// Mitsubishi GX Works2 project: GBOD-1507C(20080005)_210617up   PLC: Q03UDV

PROGRAM MAIN
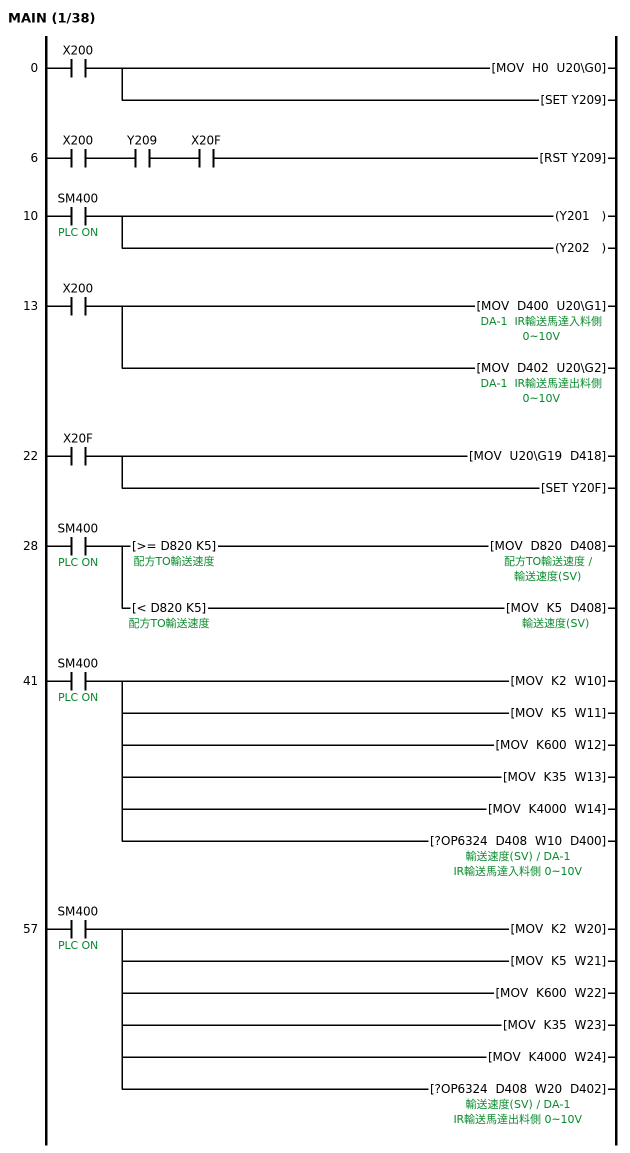
0     LD      X200
      MOV     H0 U20\G0
      SET     Y209
6     LD      X200
      AND     Y209
      AND     X20F
      RST     Y209
10    LD      SM400  ; PLC ON
      OUT     Y201
      OUT     Y202
13    LD      X200
      MOV     D400 U20\G1  ; DA-1  IR輸送馬達入料側 0~10V
      MOV     D402 U20\G2  ; DA-1  IR輸送馬達出料側 0~10V
22    LD      X20F
      MOV     U20\G19 D418
      SET     Y20F
28    LD      SM400  ; PLC ON
      MPS
      AND>=   D820 K5  ; 配方TO輸送速度
      MOV     D820 D408  ; 輸送速度(SV)
      MPP
      AND<    D820 K5  ; 配方TO輸送速度
      MOV     K5 D408
41    LD      SM400  ; PLC ON
      MOV     K2 W10
        [note] 
      MOV     K5 W11
      MOV     K600 W12
      MOV     K35 W13
      MOV     K4000 W14
      ?OP6324 D408 W10 D400
57    LD      SM400  ; PLC ON
      MOV     K2 W20
        [note] 
      MOV     K5 W21
      MOV     K600 W22
      MOV     K35 W23
      MOV     K4000 W24
      ?OP6324 D408 W20 D402
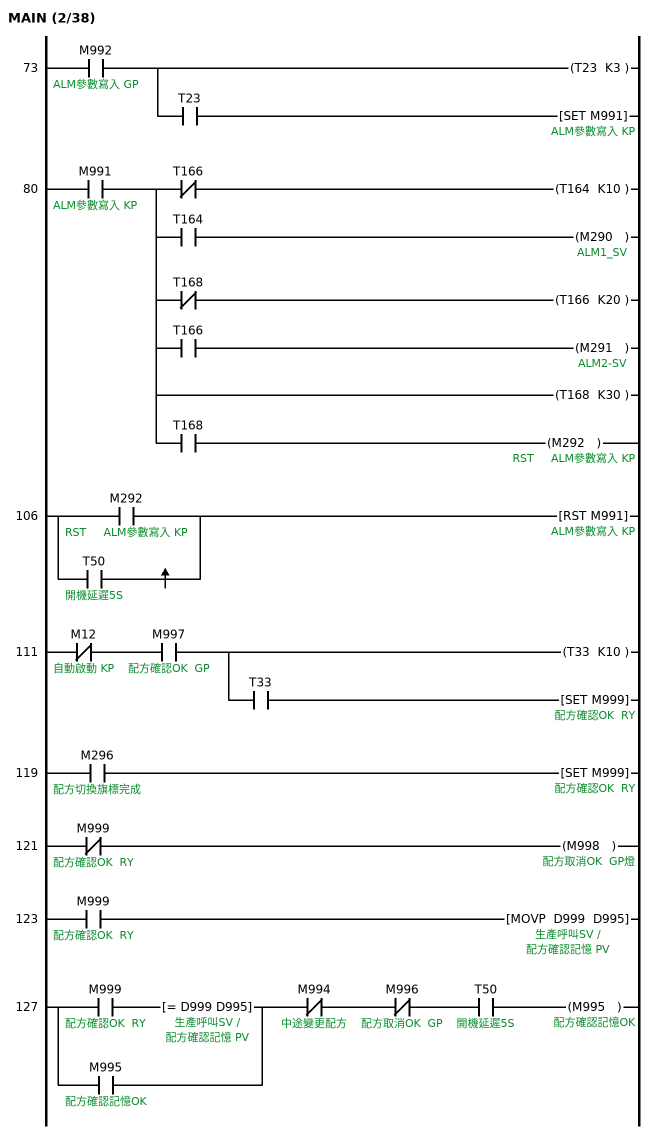
73    LD      M992  ; ALM參數寫入 GP
      OUT     T23 K3
      AND     T23
      SET     M991  ; ALM參數寫入 KP
80    LD      M991  ; ALM參數寫入 KP
      MPS
      ANI     T166
      OUT     T164 K10
      MRD
      AND     T164
      OUT     M290  ; ALM1_SV
      MRD
      ANI     T168
      OUT     T166 K20
      MRD
      AND     T166
      OUT     M291  ; ALM2-SV
      MPP
      OUT     T168 K30
      AND     T168
      OUT     M292  ; RST     ALM參數寫入 KP
106   LD      M292  ; RST     ALM參數寫入 KP
      LD      T50  ; 開機延遲5S
      MEP
      ORB
      RST     M991  ; ALM參數寫入 KP
111   LDI     M12  ; 自動啟動 KP
      AND     M997  ; 配方確認OK  GP
      OUT     T33 K10
      AND     T33
      SET     M999  ; 配方確認OK  RY
119   LD      M296  ; 配方切換旗標完成
      SET     M999  ; 配方確認OK  RY
121   LDI     M999  ; 配方確認OK  RY
      OUT     M998  ; 配方取消OK  GP燈
123   LD      M999  ; 配方確認OK  RY
      MOVP    D999 D995  ; 生產呼叫SV / 配方確認記憶 PV
127   LD      M999  ; 配方確認OK  RY
      AND=    D999 D995  ; 生產呼叫SV / 配方確認記憶 PV
      OR      M995  ; 配方確認記憶OK
      ANI     M994  ; 中途變更配方
      ANI     M996  ; 配方取消OK  GP
      AND     T50  ; 開機延遲5S
      OUT     M995  ; 配方確認記憶OK
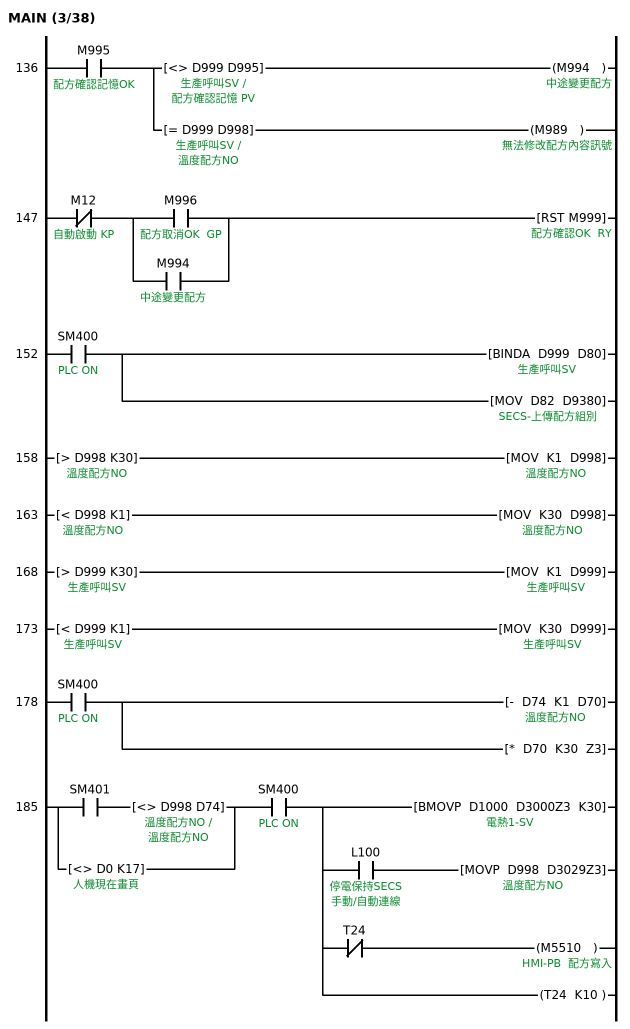
136   LD      M995  ; 配方確認記憶OK
      MPS
      AND<>   D999 D995  ; 生產呼叫SV / 配方確認記憶 PV
      OUT     M994  ; 中途變更配方
      MPP
      AND=    D999 D998  ; 生產呼叫SV / 溫度配方NO
      OUT     M989  ; 無法修改配方內容訊號
147   LDI     M12  ; 自動啟動 KP
      LD      M996  ; 配方取消OK  GP
      OR      M994  ; 中途變更配方
      ANB
      RST     M999  ; 配方確認OK  RY
152   LD      SM400  ; PLC ON
      BINDA   D999 D80
      MOV     D82 D9380  ; SECS-上傳配方組別
158   LD>     D998 K30  ; 溫度配方NO
      MOV     K1 D998
163   LD<     D998 K1  ; 溫度配方NO
      MOV     K30 D998
168   LD>     D999 K30  ; 生產呼叫SV
      MOV     K1 D999
173   LD<     D999 K1  ; 生產呼叫SV
      MOV     K30 D999
178   LD      SM400  ; PLC ON
      -       D74 K1 D70  ; 溫度配方NO
      *       D70 K30 Z3
185   LD      SM401
      AND<>   D998 D74  ; 溫度配方NO / 溫度配方NO
      OR<>    D0 K17  ; 人機現在畫頁
      AND     SM400  ; PLC ON
      BMOVP   D1000 D3000Z3 K30  ; 電熱1-SV
      MPS
      AND     L100  ; 停電保持SECS    手動/自動連線
      MOVP    D998 D3029Z3
      MRD
      ANI     T24
      OUT     M5510  ; HMI-PB  配方寫入
      MPP
      OUT     T24 K10
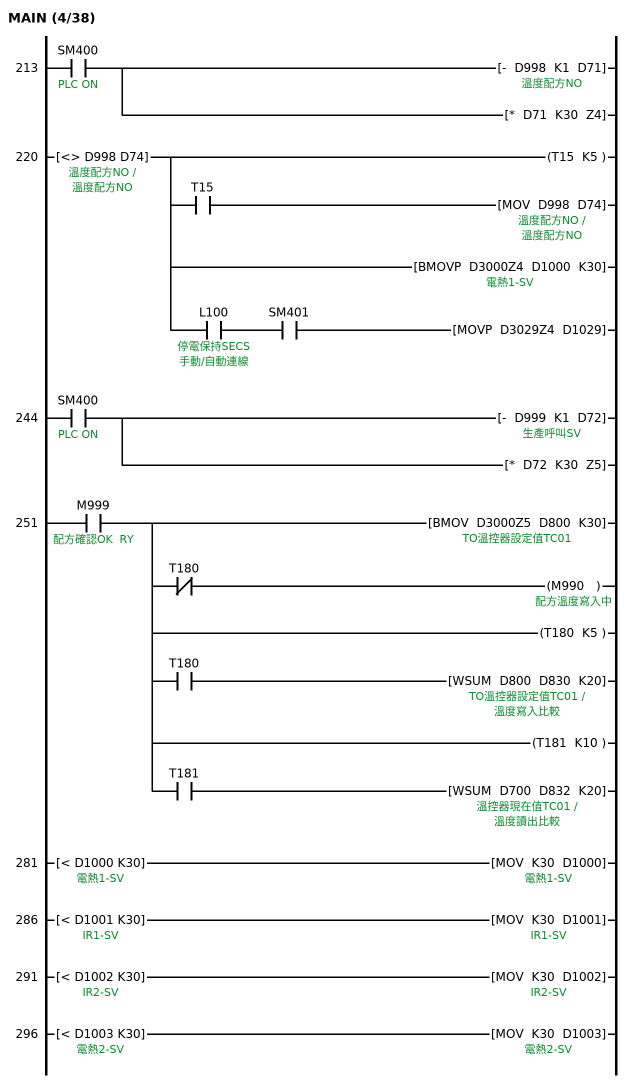
213   LD      SM400  ; PLC ON
      -       D998 K1 D71
      *       D71 K30 Z4
220   LD<>    D998 D74  ; 溫度配方NO / 溫度配方NO
      OUT     T15 K5
      MPS
      AND     T15
      MOV     D998 D74
      MPP
      BMOVP   D3000Z4 D1000 K30
      AND     L100  ; 停電保持SECS    手動/自動連線
      AND     SM401
      MOVP    D3029Z4 D1029
244   LD      SM400  ; PLC ON
      -       D999 K1 D72
      *       D72 K30 Z5
251   LD      M999  ; 配方確認OK  RY
      BMOV    D3000Z5 D800 K30  ; TO溫控器設定值TC01
      MPS
      ANI     T180
      OUT     M990  ; 配方溫度寫入中
      MPP
      OUT     T180 K5
      MPS
      AND     T180
      WSUM    D800 D830 K20  ; 溫度寫入比較
      MPP
      OUT     T181 K10
      AND     T181
      WSUM    D700 D832 K20  ; 溫控器現在值TC01 / 溫度讀出比較
281   LD<     D1000 K30  ; 電熱1-SV
      MOV     K30 D1000
286   LD<     D1001 K30  ; IR1-SV
      MOV     K30 D1001
291   LD<     D1002 K30  ; IR2-SV
      MOV     K30 D1002
296   LD<     D1003 K30  ; 電熱2-SV
      MOV     K30 D1003
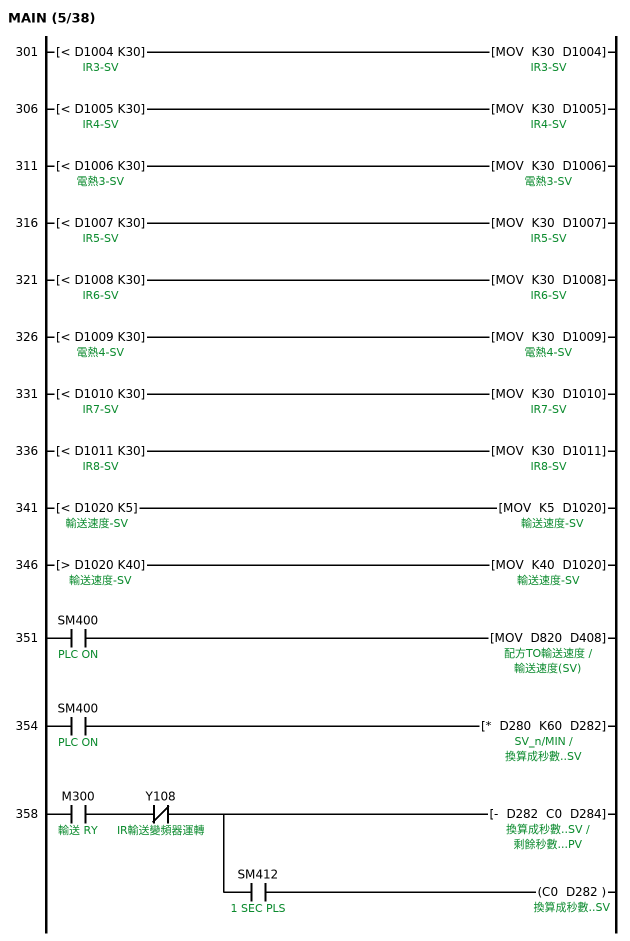
301   LD<     D1004 K30  ; IR3-SV
      MOV     K30 D1004
306   LD<     D1005 K30  ; IR4-SV
      MOV     K30 D1005
311   LD<     D1006 K30  ; 電熱3-SV
      MOV     K30 D1006
316   LD<     D1007 K30  ; IR5-SV
      MOV     K30 D1007
321   LD<     D1008 K30  ; IR6-SV
      MOV     K30 D1008
326   LD<     D1009 K30  ; 電熱4-SV
      MOV     K30 D1009
331   LD<     D1010 K30  ; IR7-SV
      MOV     K30 D1010
336   LD<     D1011 K30  ; IR8-SV
      MOV     K30 D1011
341   LD<     D1020 K5  ; 輸送速度-SV
      MOV     K5 D1020
346   LD>     D1020 K40  ; 輸送速度-SV
      MOV     K40 D1020
351   LD      SM400  ; PLC ON
      MOV     D820 D408
354   LD      SM400  ; PLC ON
      *       D280 K60 D282  ; SV_n/MIN / 換算成秒數..SV
358   LD      M300  ; 輸送 RY
      ANI     Y108  ; IR輸送變頻器運轉
      -       D282 C0 D284  ; 剩餘秒數...PV
      AND     SM412  ; 1 SEC PLS
      OUT     C0 D282  ; 換算成秒數..SV
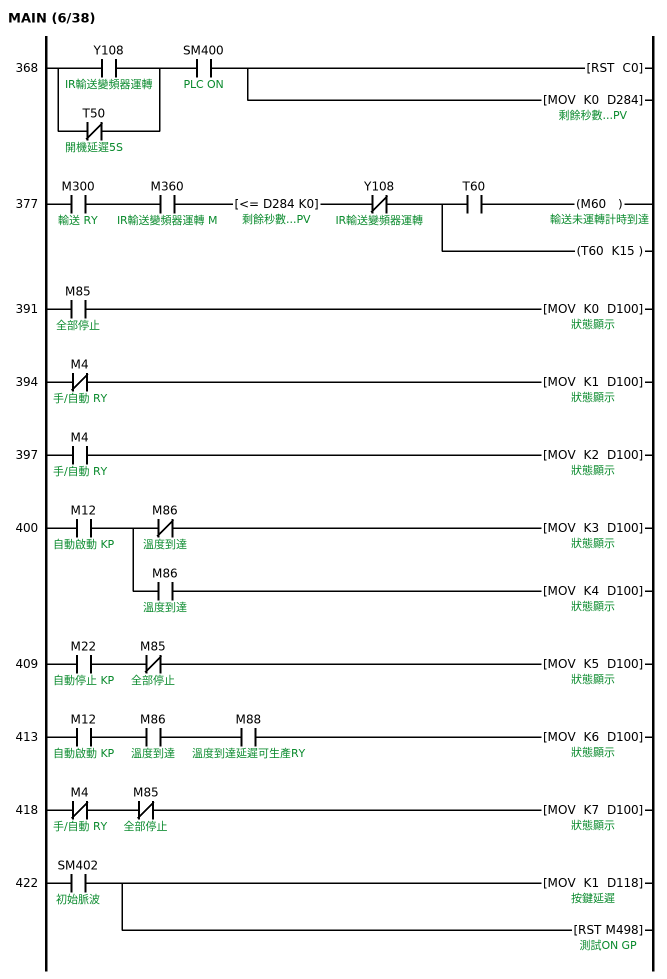
368   LD      Y108  ; IR輸送變頻器運轉
      ORI     T50  ; 開機延遲5S
      AND     SM400  ; PLC ON
      RST     C0
      MOV     K0 D284
377   LD      M300  ; 輸送 RY
      AND     M360  ; IR輸送變頻器運轉 M
      AND<=   D284 K0  ; 剩餘秒數...PV
      ANI     Y108  ; IR輸送變頻器運轉
      MPS
      AND     T60
      OUT     M60  ; 輸送未運轉計時到達
      MPP
      OUT     T60 K15
391   LD      M85  ; 全部停止
      MOV     K0 D100  ; 狀態顯示
394   LDI     M4  ; 手/自動 RY
      MOV     K1 D100
397   LD      M4  ; 手/自動 RY
      MOV     K2 D100
400   LD      M12  ; 自動啟動 KP
      MPS
      ANI     M86  ; 溫度到達
      MOV     K3 D100
      MPP
      AND     M86  ; 溫度到達
      MOV     K4 D100
409   LD      M22  ; 自動停止 KP
      ANI     M85  ; 全部停止
      MOV     K5 D100
413   LD      M12  ; 自動啟動 KP
      AND     M86  ; 溫度到達
      AND     M88  ; 溫度到達延遲可生產RY
      MOV     K6 D100
418   LDI     M4  ; 手/自動 RY
      ANI     M85  ; 全部停止
      MOV     K7 D100
422   LD      SM402  ; 初始脈波
      MOV     K1 D118  ; 按鍵延遲
      RST     M498  ; 測試ON GP
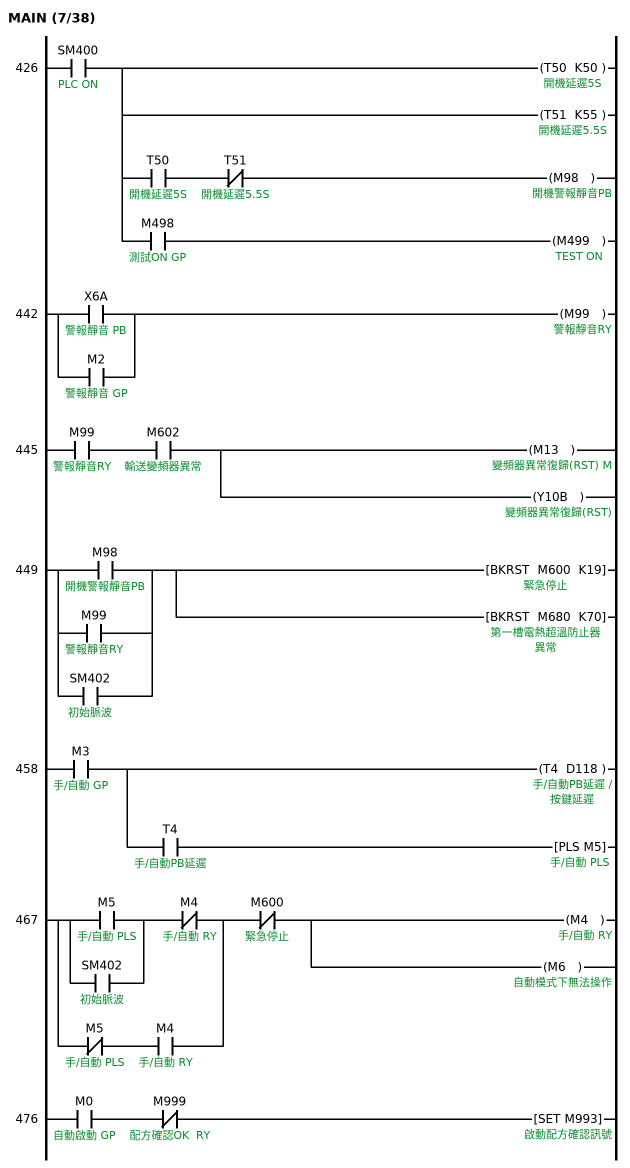
426   LD      SM400  ; PLC ON
      OUT     T50 K50  ; 開機延遲5S
      OUT     T51 K55  ; 開機延遲5.5S
      MPS
      AND     T50  ; 開機延遲5S
      ANI     T51  ; 開機延遲5.5S
      OUT     M98  ; 開機警報靜音PB
      MPP
      AND     M498  ; 測試ON GP
      OUT     M499  ; TEST ON
442   LD      X6A  ; 警報靜音 PB
      OR      M2  ; 警報靜音 GP
      OUT     M99  ; 警報靜音RY
445   LD      M99  ; 警報靜音RY
      AND     M602  ; 輸送變頻器異常
      OUT     M13  ; 變頻器異常復歸(RST) M
      OUT     Y10B  ; 變頻器異常復歸(RST)
449   LD      M98  ; 開機警報靜音PB
      OR      M99  ; 警報靜音RY
      OR      SM402  ; 初始脈波
      BKRST   M600 K19  ; 緊急停止
      BKRST   M680 K70  ; 第一槽電熱超溫防止器異常
458   LD      M3  ; 手/自動 GP
      OUT     T4 D118  ; 手/自動PB延遲 / 按鍵延遲
        [note] 
      AND     T4  ; 手/自動PB延遲
      PLS     M5  ; 手/自動 PLS
467   LD      M5  ; 手/自動 PLS
      OR      SM402  ; 初始脈波
      ANI     M4  ; 手/自動 RY
      LDI     M5  ; 手/自動 PLS
      AND     M4  ; 手/自動 RY
      ORB
      ANI     M600  ; 緊急停止
      OUT     M4  ; 手/自動 RY
      OUT     M6  ; 自動模式下無法操作
476   LD      M0  ; 自動啟動 GP
      ANI     M999  ; 配方確認OK  RY
      SET     M993  ; 啟動配方確認訊號
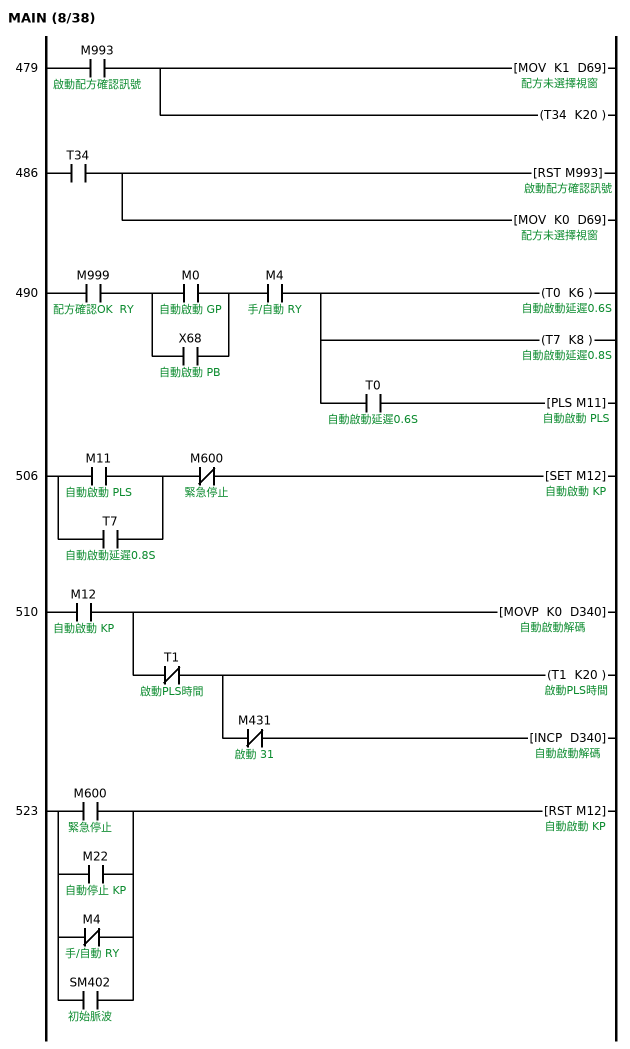
479   LD      M993  ; 啟動配方確認訊號
      MOV     K1 D69  ; 配方未選擇視窗
      OUT     T34 K20
486   LD      T34
      RST     M993  ; 啟動配方確認訊號
      MOV     K0 D69
490   LD      M999  ; 配方確認OK  RY
      LD      M0  ; 自動啟動 GP
      OR      X68  ; 自動啟動 PB
      ANB
      AND     M4  ; 手/自動 RY
      OUT     T0 K6  ; 自動啟動延遲0.6S
      OUT     T7 K8  ; 自動啟動延遲0.8S
      AND     T0  ; 自動啟動延遲0.6S
      PLS     M11  ; 自動啟動 PLS
506   LD      M11  ; 自動啟動 PLS
      OR      T7  ; 自動啟動延遲0.8S
      ANI     M600  ; 緊急停止
      SET     M12  ; 自動啟動 KP
510   LD      M12  ; 自動啟動 KP
      MOVP    K0 D340  ; 自動啟動解碼
      ANI     T1  ; 啟動PLS時間
      OUT     T1 K20  ; 啟動PLS時間
      ANI     M431  ; 啟動 31
      INCP    D340
523   LD      M600  ; 緊急停止
      OR      M22  ; 自動停止 KP
      ORI     M4  ; 手/自動 RY
      OR      SM402  ; 初始脈波
      RST     M12  ; 自動啟動 KP
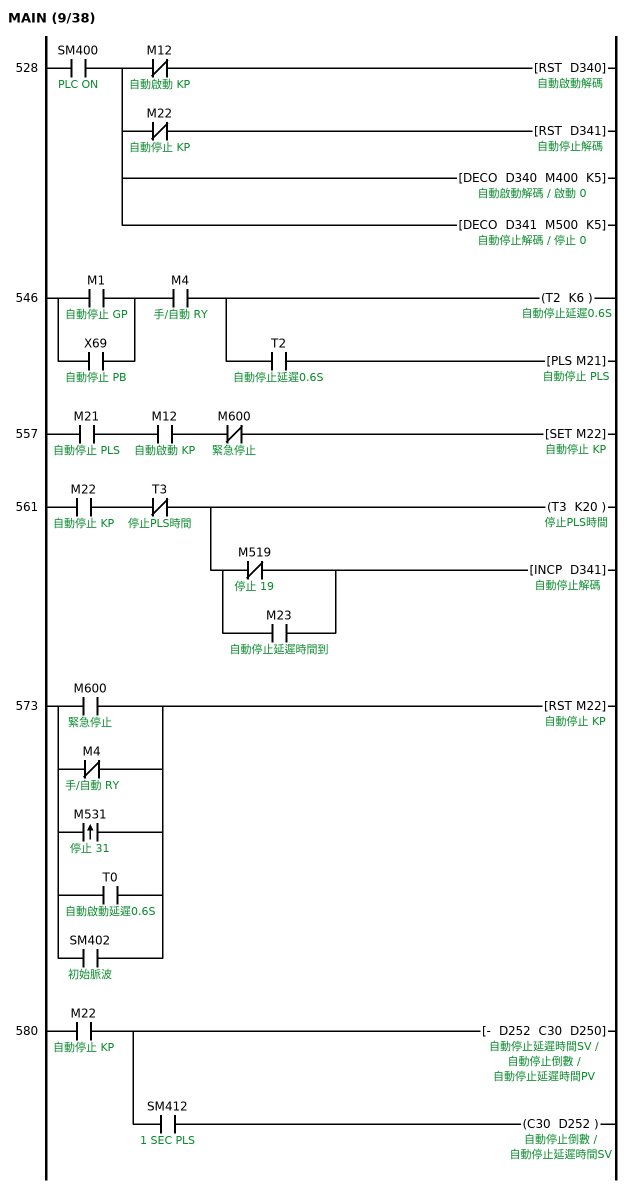
528   LD      SM400  ; PLC ON
      MPS
      ANI     M12  ; 自動啟動 KP
      RST     D340  ; 自動啟動解碼
      MRD
      ANI     M22  ; 自動停止 KP
      RST     D341  ; 自動停止解碼
      MPP
      DECO    D340 M400 K5  ; 啟動 0
      DECO    D341 M500 K5  ; 停止 0
546   LD      M1  ; 自動停止 GP
      OR      X69  ; 自動停止 PB
      AND     M4  ; 手/自動 RY
      OUT     T2 K6  ; 自動停止延遲0.6S
        [note] 
      AND     T2  ; 自動停止延遲0.6S
      PLS     M21  ; 自動停止 PLS
557   LD      M21  ; 自動停止 PLS
      AND     M12  ; 自動啟動 KP
      ANI     M600  ; 緊急停止
      SET     M22  ; 自動停止 KP
561   LD      M22  ; 自動停止 KP
      ANI     T3  ; 停止PLS時間
      OUT     T3 K20  ; 停止PLS時間
      LDI     M519  ; 停止 19
      OR      M23  ; 自動停止延遲時間到
      ANB
      INCP    D341
573   LD      M600  ; 緊急停止
      ORI     M4  ; 手/自動 RY
      ORP     M531  ; 停止 31
      OR      T0  ; 自動啟動延遲0.6S
      OR      SM402  ; 初始脈波
      RST     M22  ; 自動停止 KP
580   LD      M22  ; 自動停止 KP
      -       D252 C30 D250  ; 自動停止延遲時間SV / 自動停止倒數 / 自動停止延遲時間PV
      AND     SM412  ; 1 SEC PLS
      OUT     C30 D252  ; 自動停止倒數 / 自動停止延遲時間SV
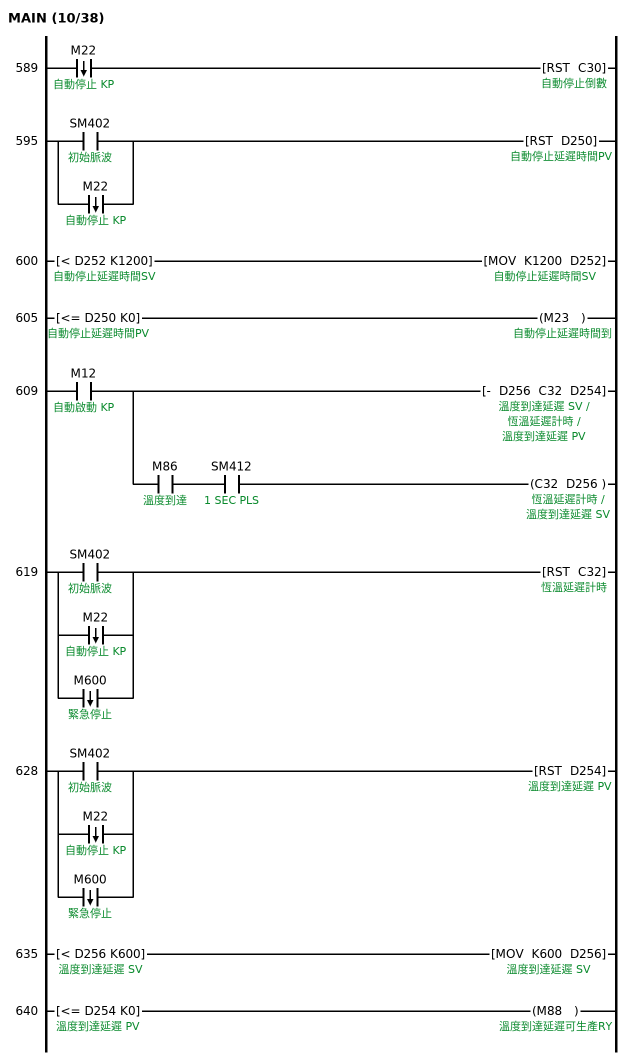
589   LDF     M22  ; 自動停止 KP
      RST     C30  ; 自動停止倒數
595   LD      SM402  ; 初始脈波
      ORF     M22  ; 自動停止 KP
      RST     D250  ; 自動停止延遲時間PV
600   LD<     D252 K1200  ; 自動停止延遲時間SV
      MOV     K1200 D252
605   LD<=    D250 K0  ; 自動停止延遲時間PV
      OUT     M23  ; 自動停止延遲時間到
609   LD      M12  ; 自動啟動 KP
      -       D256 C32 D254  ; 溫度到達延遲 SV / 恆溫延遲計時 / 溫度到達延遲 PV
      AND     M86  ; 溫度到達
      AND     SM412  ; 1 SEC PLS
      OUT     C32 D256  ; 恆溫延遲計時 / 溫度到達延遲 SV
619   LD      SM402  ; 初始脈波
      ORF     M22  ; 自動停止 KP
      ORF     M600  ; 緊急停止
      RST     C32  ; 恆溫延遲計時
628   LD      SM402  ; 初始脈波
      ORF     M22  ; 自動停止 KP
      ORF     M600  ; 緊急停止
      RST     D254  ; 溫度到達延遲 PV
635   LD<     D256 K600  ; 溫度到達延遲 SV
      MOV     K600 D256
640   LD<=    D254 K0  ; 溫度到達延遲 PV
      OUT     M88  ; 溫度到達延遲可生產RY
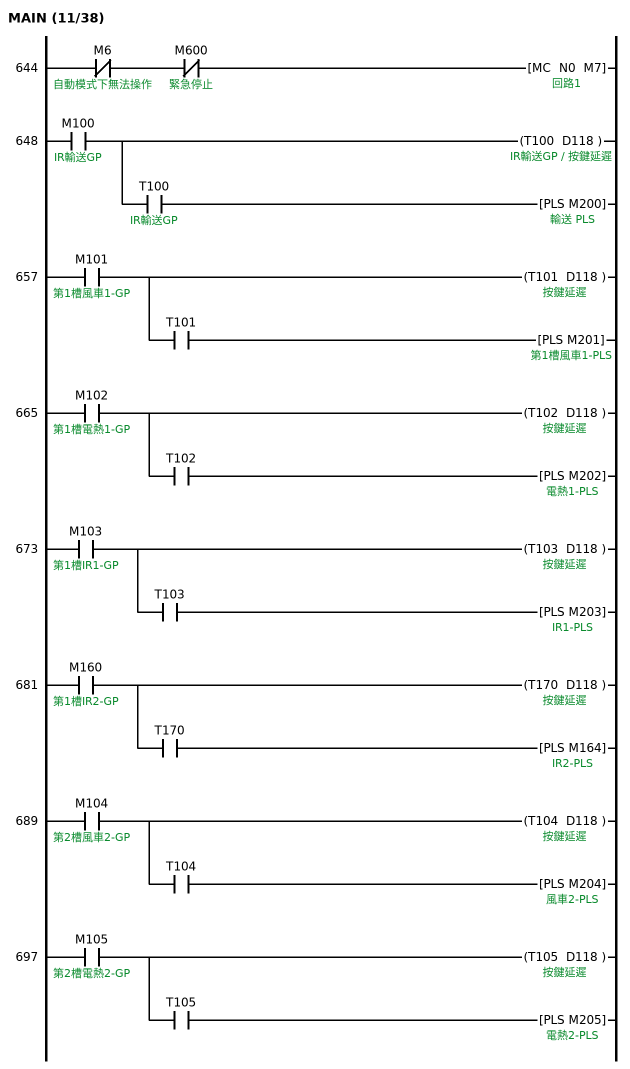
644   LDI     M6  ; 自動模式下無法操作
      ANI     M600  ; 緊急停止
      MC      N0 M7  ; 回路1
648   LD      M100  ; IR輸送GP
      OUT     T100 D118  ; IR輸送GP / 按鍵延遲
        [note] 
      AND     T100  ; IR輸送GP
      PLS     M200  ; 輸送 PLS
657   LD      M101  ; 第1槽風車1-GP
      OUT     T101 D118  ; 按鍵延遲
      AND     T101
      PLS     M201  ; 第1槽風車1-PLS
665   LD      M102  ; 第1槽電熱1-GP
      OUT     T102 D118  ; 按鍵延遲
      AND     T102
      PLS     M202  ; 電熱1-PLS
673   LD      M103  ; 第1槽IR1-GP
      OUT     T103 D118  ; 按鍵延遲
      AND     T103
      PLS     M203  ; IR1-PLS
681   LD      M160  ; 第1槽IR2-GP
      OUT     T170 D118  ; 按鍵延遲
      AND     T170
      PLS     M164  ; IR2-PLS
689   LD      M104  ; 第2槽風車2-GP
      OUT     T104 D118  ; 按鍵延遲
      AND     T104
      PLS     M204  ; 風車2-PLS
697   LD      M105  ; 第2槽電熱2-GP
      OUT     T105 D118  ; 按鍵延遲
      AND     T105
      PLS     M205  ; 電熱2-PLS
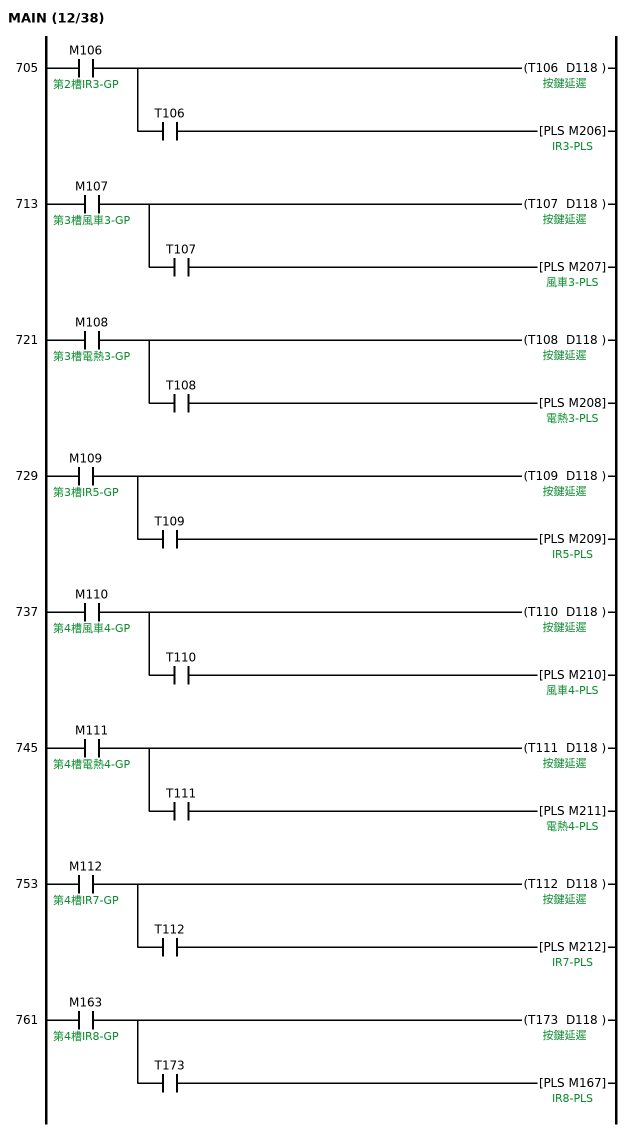
705   LD      M106  ; 第2槽IR3-GP
      OUT     T106 D118  ; 按鍵延遲
      AND     T106
      PLS     M206  ; IR3-PLS
713   LD      M107  ; 第3槽風車3-GP
      OUT     T107 D118  ; 按鍵延遲
      AND     T107
      PLS     M207  ; 風車3-PLS
721   LD      M108  ; 第3槽電熱3-GP
      OUT     T108 D118  ; 按鍵延遲
      AND     T108
      PLS     M208  ; 電熱3-PLS
729   LD      M109  ; 第3槽IR5-GP
      OUT     T109 D118  ; 按鍵延遲
      AND     T109
      PLS     M209  ; IR5-PLS
737   LD      M110  ; 第4槽風車4-GP
      OUT     T110 D118  ; 按鍵延遲
      AND     T110
      PLS     M210  ; 風車4-PLS
745   LD      M111  ; 第4槽電熱4-GP
      OUT     T111 D118  ; 按鍵延遲
      AND     T111
      PLS     M211  ; 電熱4-PLS
753   LD      M112  ; 第4槽IR7-GP
      OUT     T112 D118  ; 按鍵延遲
      AND     T112
      PLS     M212  ; IR7-PLS
761   LD      M163  ; 第4槽IR8-GP
      OUT     T173 D118  ; 按鍵延遲
      AND     T173
      PLS     M167  ; IR8-PLS
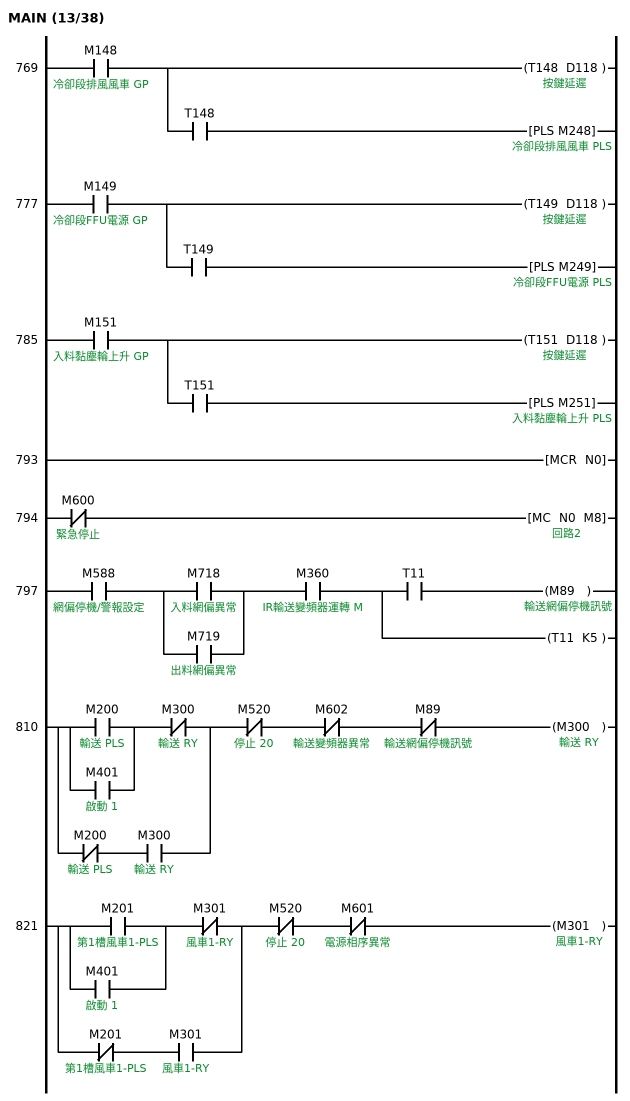
769   LD      M148  ; 冷卻段排風風車 GP
      OUT     T148 D118  ; 按鍵延遲
      AND     T148
      PLS     M248  ; 冷卻段排風風車 PLS
777   LD      M149  ; 冷卻段FFU電源 GP
      OUT     T149 D118  ; 按鍵延遲
      AND     T149
      PLS     M249  ; 冷卻段FFU電源 PLS
785   LD      M151  ; 入料黏塵輪上升 GP
      OUT     T151 D118  ; 按鍵延遲
      AND     T151
      PLS     M251  ; 入料黏塵輪上升 PLS
793   MCR     N0
794   LDI     M600  ; 緊急停止
      MC      N0 M8  ; 回路2
797   LD      M588  ; 網偏停機/警報設定
      LD      M718  ; 入料網偏異常
      OR      M719  ; 出料網偏異常
      ANB
      AND     M360  ; IR輸送變頻器運轉 M
      MPS
      AND     T11
      OUT     M89  ; 輸送網偏停機訊號
      MPP
      OUT     T11 K5
810   LD      M200  ; 輸送 PLS
      OR      M401  ; 啟動 1
      ANI     M300  ; 輸送 RY
      LDI     M200  ; 輸送 PLS
      AND     M300  ; 輸送 RY
      ORB
      ANI     M520  ; 停止 20
      ANI     M602  ; 輸送變頻器異常
      ANI     M89  ; 輸送網偏停機訊號
      OUT     M300  ; 輸送 RY
        [note] 
821   LD      M201  ; 第1槽風車1-PLS
      OR      M401  ; 啟動 1
      ANI     M301  ; 風車1-RY
      LDI     M201  ; 第1槽風車1-PLS
      AND     M301  ; 風車1-RY
      ORB
      ANI     M520  ; 停止 20
      ANI     M601  ; 電源相序異常
      OUT     M301  ; 風車1-RY
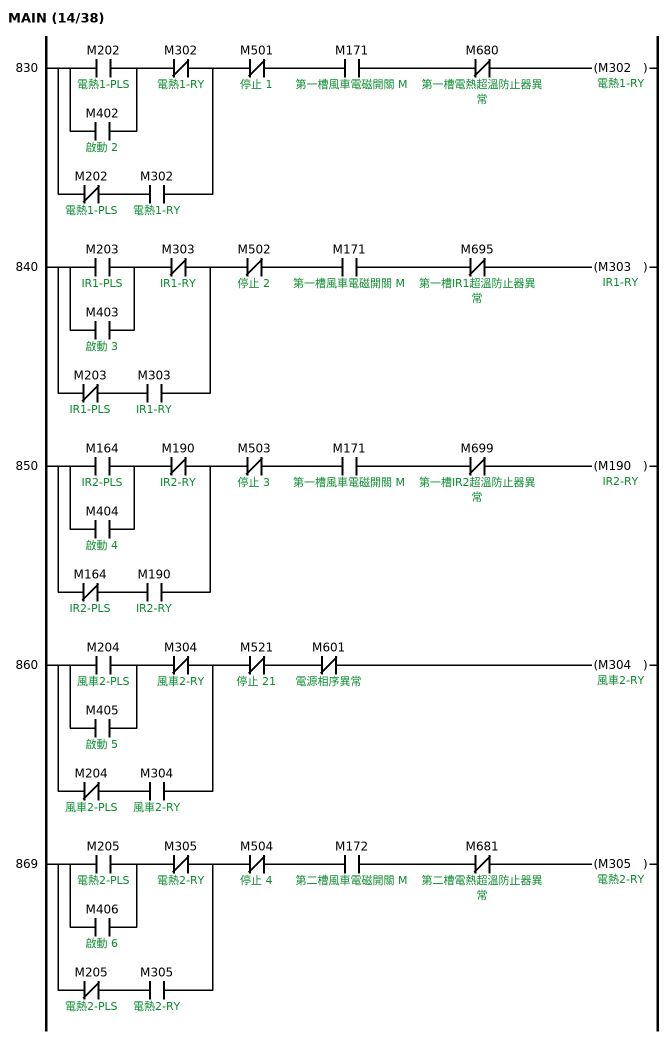
830   LD      M202  ; 電熱1-PLS
      OR      M402  ; 啟動 2
      ANI     M302  ; 電熱1-RY
      LDI     M202  ; 電熱1-PLS
      AND     M302  ; 電熱1-RY
      ORB
      ANI     M501  ; 停止 1
      AND     M171  ; 第一槽風車電磁開關 M
      ANI     M680  ; 第一槽電熱超溫防止器異常
      OUT     M302  ; 電熱1-RY
840   LD      M203  ; IR1-PLS
      OR      M403  ; 啟動 3
      ANI     M303  ; IR1-RY
      LDI     M203  ; IR1-PLS
      AND     M303  ; IR1-RY
      ORB
      ANI     M502  ; 停止 2
      AND     M171  ; 第一槽風車電磁開關 M
      ANI     M695  ; 第一槽IR1超溫防止器異常
      OUT     M303  ; IR1-RY
850   LD      M164  ; IR2-PLS
      OR      M404  ; 啟動 4
      ANI     M190  ; IR2-RY
      LDI     M164  ; IR2-PLS
      AND     M190  ; IR2-RY
      ORB
      ANI     M503  ; 停止 3
      AND     M171  ; 第一槽風車電磁開關 M
      ANI     M699  ; 第一槽IR2超溫防止器異常
      OUT     M190  ; IR2-RY
860   LD      M204  ; 風車2-PLS
      OR      M405  ; 啟動 5
      ANI     M304  ; 風車2-RY
      LDI     M204  ; 風車2-PLS
      AND     M304  ; 風車2-RY
      ORB
      ANI     M521  ; 停止 21
      ANI     M601  ; 電源相序異常
      OUT     M304  ; 風車2-RY
869   LD      M205  ; 電熱2-PLS
      OR      M406  ; 啟動 6
      ANI     M305  ; 電熱2-RY
      LDI     M205  ; 電熱2-PLS
      AND     M305  ; 電熱2-RY
      ORB
      ANI     M504  ; 停止 4
      AND     M172  ; 第二槽風車電磁開關 M
      ANI     M681  ; 第二槽電熱超溫防止器異常
      OUT     M305  ; 電熱2-RY
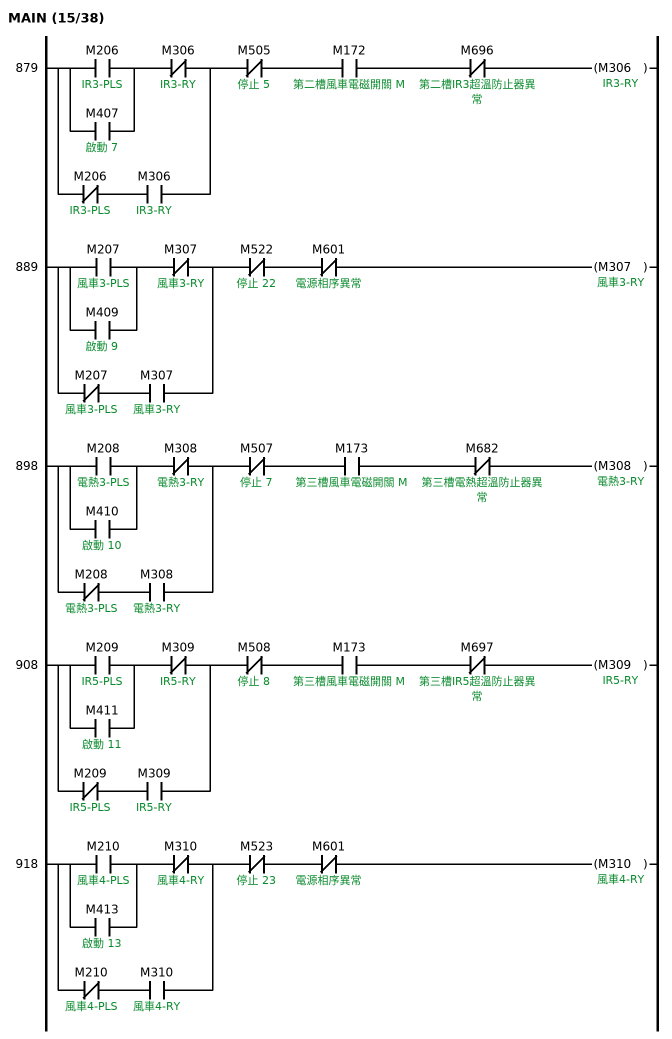
879   LD      M206  ; IR3-PLS
      OR      M407  ; 啟動 7
      ANI     M306  ; IR3-RY
      LDI     M206  ; IR3-PLS
      AND     M306  ; IR3-RY
      ORB
      ANI     M505  ; 停止 5
      AND     M172  ; 第二槽風車電磁開關 M
      ANI     M696  ; 第二槽IR3超溫防止器異常
      OUT     M306  ; IR3-RY
889   LD      M207  ; 風車3-PLS
      OR      M409  ; 啟動 9
      ANI     M307  ; 風車3-RY
      LDI     M207  ; 風車3-PLS
      AND     M307  ; 風車3-RY
      ORB
      ANI     M522  ; 停止 22
      ANI     M601  ; 電源相序異常
      OUT     M307  ; 風車3-RY
898   LD      M208  ; 電熱3-PLS
      OR      M410  ; 啟動 10
      ANI     M308  ; 電熱3-RY
      LDI     M208  ; 電熱3-PLS
      AND     M308  ; 電熱3-RY
      ORB
      ANI     M507  ; 停止 7
      AND     M173  ; 第三槽風車電磁開關 M
      ANI     M682  ; 第三槽電熱超溫防止器異常
      OUT     M308  ; 電熱3-RY
908   LD      M209  ; IR5-PLS
      OR      M411  ; 啟動 11
      ANI     M309  ; IR5-RY
      LDI     M209  ; IR5-PLS
      AND     M309  ; IR5-RY
      ORB
      ANI     M508  ; 停止 8
      AND     M173  ; 第三槽風車電磁開關 M
      ANI     M697  ; 第三槽IR5超溫防止器異常
      OUT     M309  ; IR5-RY
918   LD      M210  ; 風車4-PLS
      OR      M413  ; 啟動 13
      ANI     M310  ; 風車4-RY
      LDI     M210  ; 風車4-PLS
      AND     M310  ; 風車4-RY
      ORB
      ANI     M523  ; 停止 23
      ANI     M601  ; 電源相序異常
      OUT     M310  ; 風車4-RY
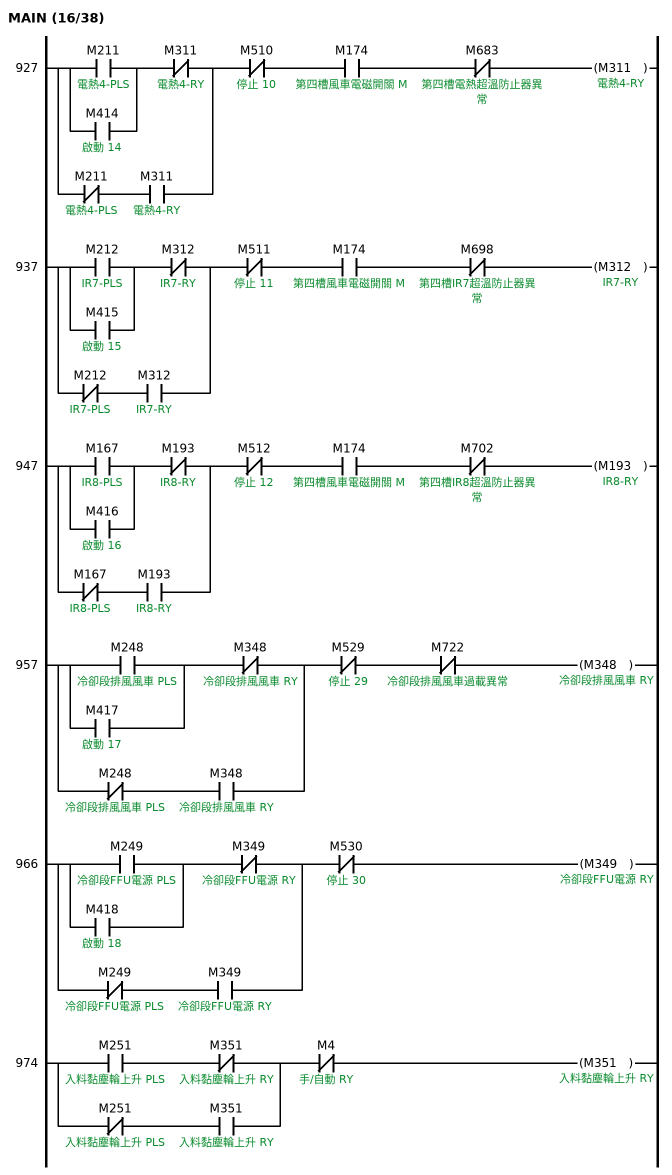
927   LD      M211  ; 電熱4-PLS
      OR      M414  ; 啟動 14
      ANI     M311  ; 電熱4-RY
      LDI     M211  ; 電熱4-PLS
      AND     M311  ; 電熱4-RY
      ORB
      ANI     M510  ; 停止 10
      AND     M174  ; 第四槽風車電磁開關 M
      ANI     M683  ; 第四槽電熱超溫防止器異常
      OUT     M311  ; 電熱4-RY
937   LD      M212  ; IR7-PLS
      OR      M415  ; 啟動 15
      ANI     M312  ; IR7-RY
      LDI     M212  ; IR7-PLS
      AND     M312  ; IR7-RY
      ORB
      ANI     M511  ; 停止 11
      AND     M174  ; 第四槽風車電磁開關 M
      ANI     M698  ; 第四槽IR7超溫防止器異常
      OUT     M312  ; IR7-RY
947   LD      M167  ; IR8-PLS
      OR      M416  ; 啟動 16
      ANI     M193  ; IR8-RY
      LDI     M167  ; IR8-PLS
      AND     M193  ; IR8-RY
      ORB
      ANI     M512  ; 停止 12
      AND     M174  ; 第四槽風車電磁開關 M
      ANI     M702  ; 第四槽IR8超溫防止器異常
      OUT     M193  ; IR8-RY
957   LD      M248  ; 冷卻段排風風車 PLS
      OR      M417  ; 啟動 17
      ANI     M348  ; 冷卻段排風風車 RY
      LDI     M248  ; 冷卻段排風風車 PLS
      AND     M348  ; 冷卻段排風風車 RY
      ORB
      ANI     M529  ; 停止 29
      ANI     M722  ; 冷卻段排風風車過載異常
      OUT     M348  ; 冷卻段排風風車 RY
966   LD      M249  ; 冷卻段FFU電源 PLS
      OR      M418  ; 啟動 18
      ANI     M349  ; 冷卻段FFU電源 RY
      LDI     M249  ; 冷卻段FFU電源 PLS
      AND     M349  ; 冷卻段FFU電源 RY
      ORB
      ANI     M530  ; 停止 30
      OUT     M349  ; 冷卻段FFU電源 RY
974   LD      M251  ; 入料黏塵輪上升 PLS
      ANI     M351  ; 入料黏塵輪上升 RY
      LDI     M251  ; 入料黏塵輪上升 PLS
      AND     M351  ; 入料黏塵輪上升 RY
      ORB
      ANI     M4  ; 手/自動 RY
      OUT     M351  ; 入料黏塵輪上升 RY
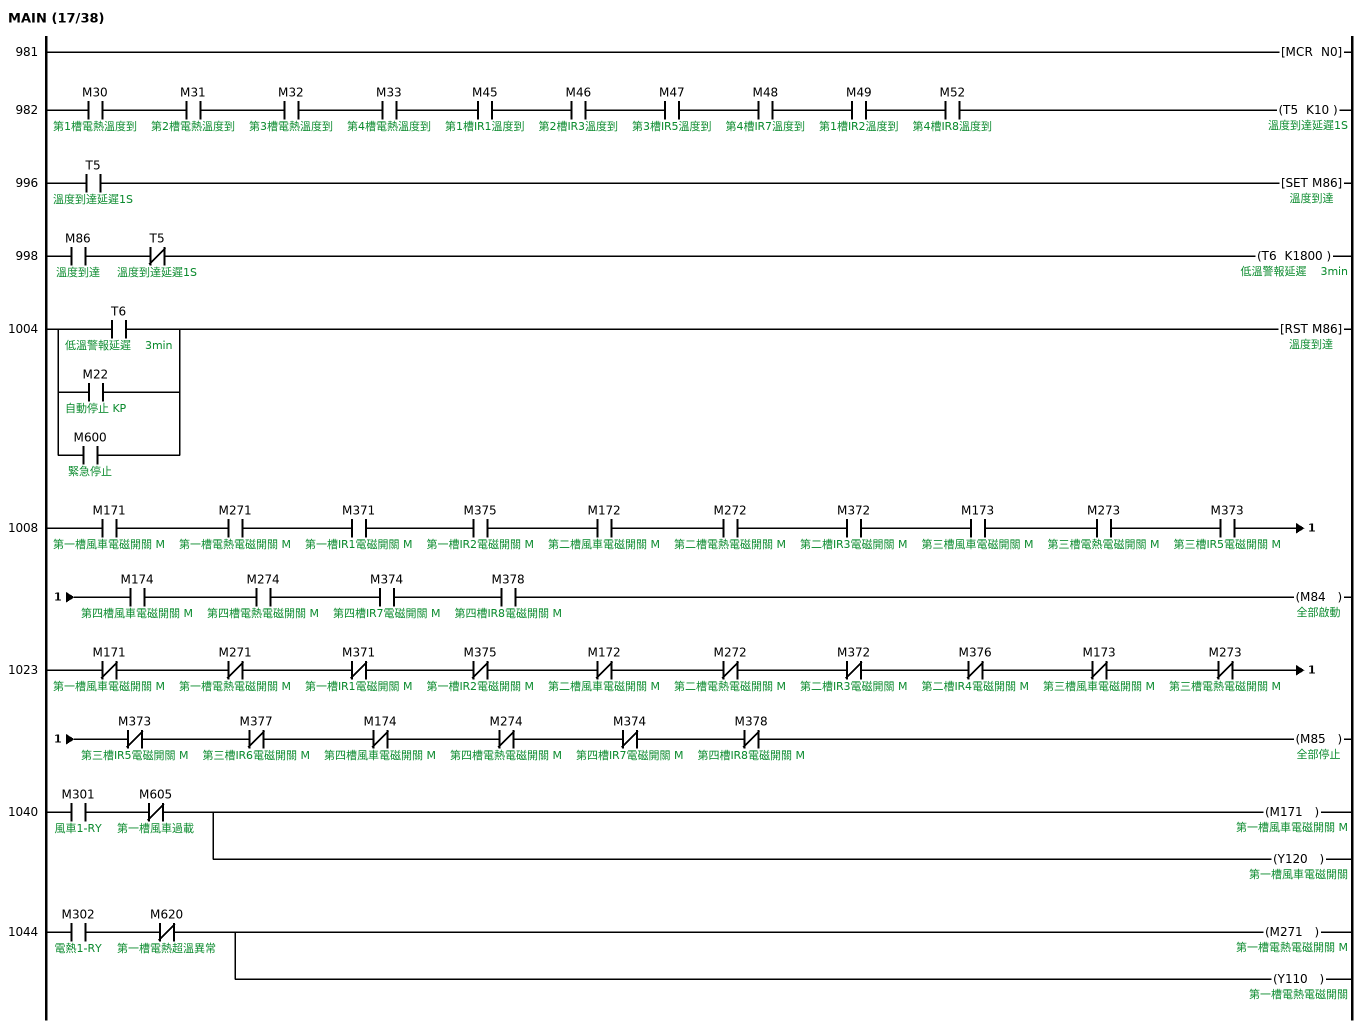
981   MCR     N0
982   LD      M30  ; 第1槽電熱溫度到
      AND     M31  ; 第2槽電熱溫度到
      AND     M32  ; 第3槽電熱溫度到
      AND     M33  ; 第4槽電熱溫度到
      AND     M45  ; 第1槽IR1溫度到
      AND     M46  ; 第2槽IR3溫度到
      AND     M47  ; 第3槽IR5溫度到
      AND     M48  ; 第4槽IR7溫度到
      AND     M49  ; 第1槽IR2溫度到
      AND     M52  ; 第4槽IR8溫度到
      OUT     T5 K10  ; 溫度到達延遲1S
996   LD      T5  ; 溫度到達延遲1S
      SET     M86  ; 溫度到達
998   LD      M86  ; 溫度到達
      ANI     T5  ; 溫度到達延遲1S
      OUT     T6 K1800  ; 低溫警報延遲    3min
1004  LD      T6  ; 低溫警報延遲    3min
      OR      M22  ; 自動停止 KP
      OR      M600  ; 緊急停止
      RST     M86  ; 溫度到達
1008  LD      M171  ; 第一槽風車電磁開關 M
      AND     M271  ; 第一槽電熱電磁開關 M
      AND     M371  ; 第一槽IR1電磁開關 M
      AND     M375  ; 第一槽IR2電磁開關 M
      AND     M172  ; 第二槽風車電磁開關 M
      AND     M272  ; 第二槽電熱電磁開關 M
      AND     M372  ; 第二槽IR3電磁開關 M
      AND     M173  ; 第三槽風車電磁開關 M
      AND     M273  ; 第三槽電熱電磁開關 M
      AND     M373  ; 第三槽IR5電磁開關 M
      AND     M174  ; 第四槽風車電磁開關 M
      AND     M274  ; 第四槽電熱電磁開關 M
      AND     M374  ; 第四槽IR7電磁開關 M
      AND     M378  ; 第四槽IR8電磁開關 M
      OUT     M84  ; 全部啟動
1023  LDI     M171  ; 第一槽風車電磁開關 M
      ANI     M271  ; 第一槽電熱電磁開關 M
      ANI     M371  ; 第一槽IR1電磁開關 M
      ANI     M375  ; 第一槽IR2電磁開關 M
      ANI     M172  ; 第二槽風車電磁開關 M
      ANI     M272  ; 第二槽電熱電磁開關 M
      ANI     M372  ; 第二槽IR3電磁開關 M
      ANI     M376  ; 第二槽IR4電磁開關 M
      ANI     M173  ; 第三槽風車電磁開關 M
      ANI     M273  ; 第三槽電熱電磁開關 M
      ANI     M373  ; 第三槽IR5電磁開關 M
      ANI     M377  ; 第三槽IR6電磁開關 M
      ANI     M174  ; 第四槽風車電磁開關 M
      ANI     M274  ; 第四槽電熱電磁開關 M
      ANI     M374  ; 第四槽IR7電磁開關 M
      ANI     M378  ; 第四槽IR8電磁開關 M
      OUT     M85  ; 全部停止
1040  LD      M301  ; 風車1-RY
      ANI     M605  ; 第一槽風車過載
      OUT     M171  ; 第一槽風車電磁開關 M
      OUT     Y120  ; 第一槽風車電磁開關
1044  LD      M302  ; 電熱1-RY
      ANI     M620  ; 第一槽電熱超溫異常
      OUT     M271  ; 第一槽電熱電磁開關 M
      OUT     Y110  ; 第一槽電熱電磁開關
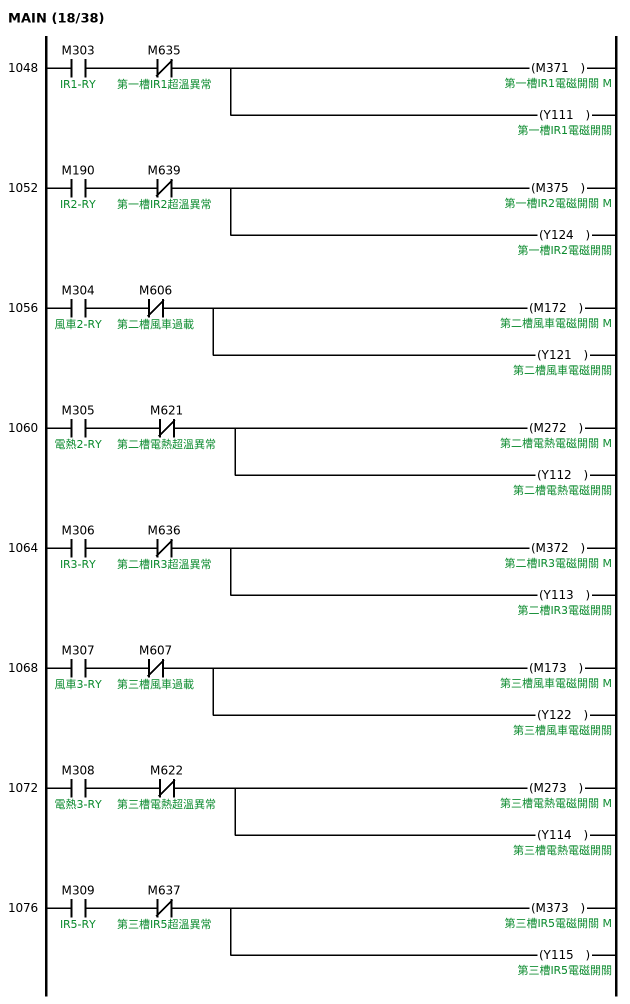
1048  LD      M303  ; IR1-RY
      ANI     M635  ; 第一槽IR1超溫異常
      OUT     M371  ; 第一槽IR1電磁開關 M
      OUT     Y111  ; 第一槽IR1電磁開關
1052  LD      M190  ; IR2-RY
      ANI     M639  ; 第一槽IR2超溫異常
      OUT     M375  ; 第一槽IR2電磁開關 M
      OUT     Y124  ; 第一槽IR2電磁開關
1056  LD      M304  ; 風車2-RY
      ANI     M606  ; 第二槽風車過載
      OUT     M172  ; 第二槽風車電磁開關 M
      OUT     Y121  ; 第二槽風車電磁開關
1060  LD      M305  ; 電熱2-RY
      ANI     M621  ; 第二槽電熱超溫異常
      OUT     M272  ; 第二槽電熱電磁開關 M
      OUT     Y112  ; 第二槽電熱電磁開關
1064  LD      M306  ; IR3-RY
      ANI     M636  ; 第二槽IR3超溫異常
      OUT     M372  ; 第二槽IR3電磁開關 M
      OUT     Y113  ; 第二槽IR3電磁開關
1068  LD      M307  ; 風車3-RY
      ANI     M607  ; 第三槽風車過載
      OUT     M173  ; 第三槽風車電磁開關 M
      OUT     Y122  ; 第三槽風車電磁開關
1072  LD      M308  ; 電熱3-RY
      ANI     M622  ; 第三槽電熱超溫異常
      OUT     M273  ; 第三槽電熱電磁開關 M
      OUT     Y114  ; 第三槽電熱電磁開關
1076  LD      M309  ; IR5-RY
      ANI     M637  ; 第三槽IR5超溫異常
      OUT     M373  ; 第三槽IR5電磁開關 M
      OUT     Y115  ; 第三槽IR5電磁開關
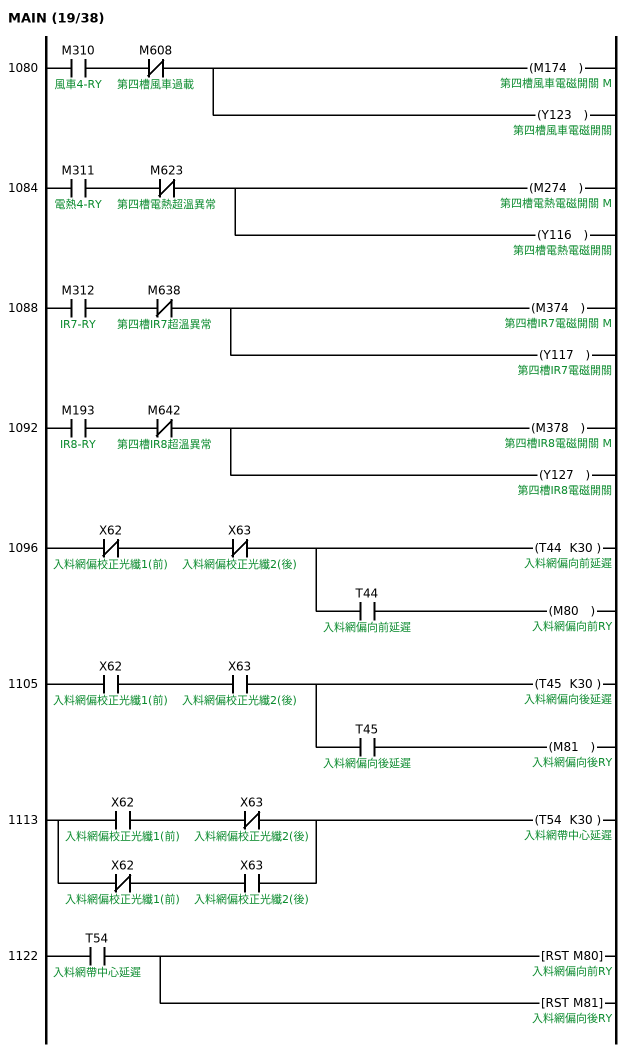
1080  LD      M310  ; 風車4-RY
      ANI     M608  ; 第四槽風車過載
      OUT     M174  ; 第四槽風車電磁開關 M
      OUT     Y123  ; 第四槽風車電磁開關
1084  LD      M311  ; 電熱4-RY
      ANI     M623  ; 第四槽電熱超溫異常
      OUT     M274  ; 第四槽電熱電磁開關 M
      OUT     Y116  ; 第四槽電熱電磁開關
1088  LD      M312  ; IR7-RY
      ANI     M638  ; 第四槽IR7超溫異常
      OUT     M374  ; 第四槽IR7電磁開關 M
      OUT     Y117  ; 第四槽IR7電磁開關
1092  LD      M193  ; IR8-RY
      ANI     M642  ; 第四槽IR8超溫異常
      OUT     M378  ; 第四槽IR8電磁開關 M
      OUT     Y127  ; 第四槽IR8電磁開關
1096  LDI     X62  ; 入料網偏校正光纖1(前)
      ANI     X63  ; 入料網偏校正光纖2(後)
      OUT     T44 K30  ; 入料網偏向前延遲
        [note] 
      AND     T44  ; 入料網偏向前延遲
      OUT     M80  ; 入料網偏向前RY
1105  LD      X62  ; 入料網偏校正光纖1(前)
      AND     X63  ; 入料網偏校正光纖2(後)
      OUT     T45 K30  ; 入料網偏向後延遲
      AND     T45  ; 入料網偏向後延遲
      OUT     M81  ; 入料網偏向後RY
1113  LD      X62  ; 入料網偏校正光纖1(前)
      ANI     X63  ; 入料網偏校正光纖2(後)
      LDI     X62  ; 入料網偏校正光纖1(前)
      AND     X63  ; 入料網偏校正光纖2(後)
      ORB
      OUT     T54 K30  ; 入料網帶中心延遲
1122  LD      T54  ; 入料網帶中心延遲
      RST     M80  ; 入料網偏向前RY
      RST     M81  ; 入料網偏向後RY
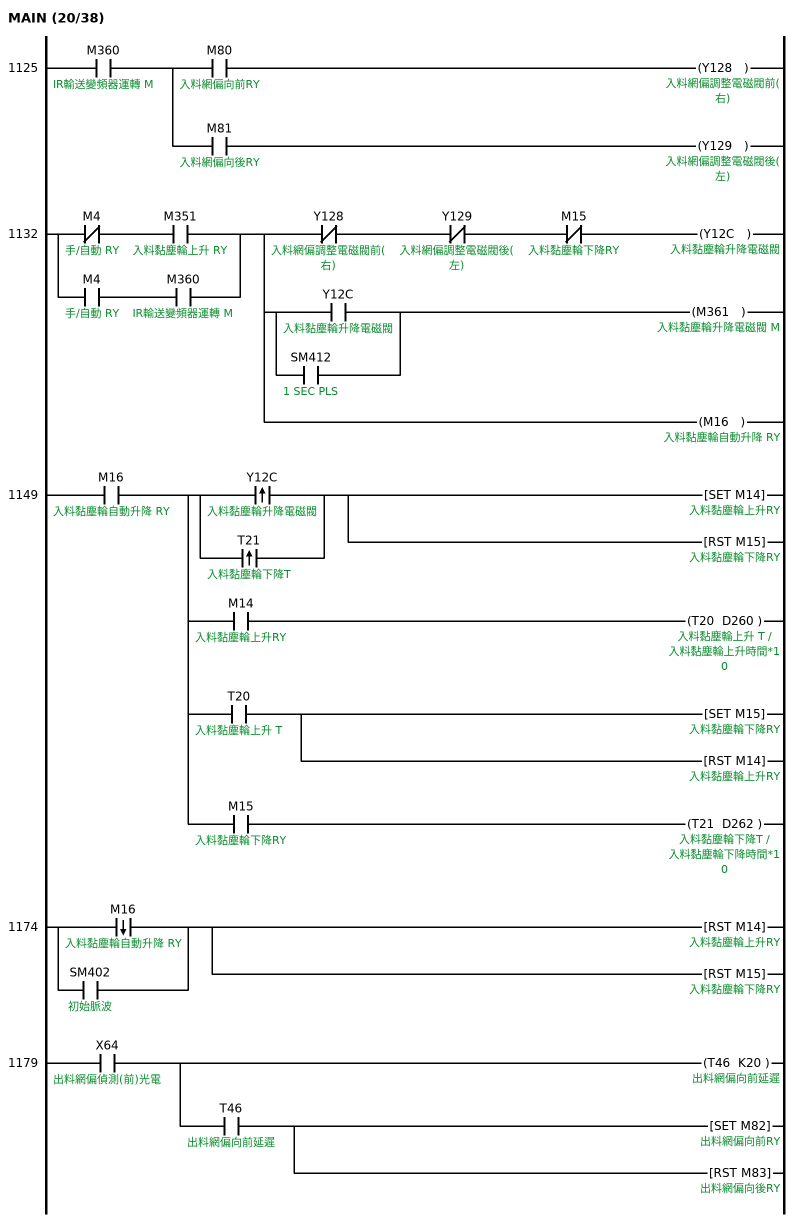
1125  LD      M360  ; IR輸送變頻器運轉 M
      MPS
      AND     M80  ; 入料網偏向前RY
      OUT     Y128  ; 入料網偏調整電磁閥前(右)
      MPP
      AND     M81  ; 入料網偏向後RY
      OUT     Y129  ; 入料網偏調整電磁閥後(左)
1132  LDI     M4  ; 手/自動 RY
      AND     M351  ; 入料黏塵輪上升 RY
      LD      M4  ; 手/自動 RY
      AND     M360  ; IR輸送變頻器運轉 M
      ORB
      MPS
      ANI     Y128  ; 入料網偏調整電磁閥前(右)
      ANI     Y129  ; 入料網偏調整電磁閥後(左)
      ANI     M15  ; 入料黏塵輪下降RY
      OUT     Y12C  ; 入料黏塵輪升降電磁閥
      MRD
      LD      Y12C  ; 入料黏塵輪升降電磁閥
      OR      SM412  ; 1 SEC PLS
      ANB
      OUT     M361  ; 入料黏塵輪升降電磁閥 M
      MPP
      OUT     M16  ; 入料黏塵輪自動升降 RY
1149  LD      M16  ; 入料黏塵輪自動升降 RY
      MPS
      LDP     Y12C  ; 入料黏塵輪升降電磁閥
      ORP     T21  ; 入料黏塵輪下降T
      ANB
      SET     M14  ; 入料黏塵輪上升RY
      RST     M15  ; 入料黏塵輪下降RY
      MRD
      AND     M14  ; 入料黏塵輪上升RY
      OUT     T20 D260  ; 入料黏塵輪上升 T / 入料黏塵輪上升時間*10
      MRD
      AND     T20  ; 入料黏塵輪上升 T
      SET     M15  ; 入料黏塵輪下降RY
      RST     M14  ; 入料黏塵輪上升RY
      MPP
      AND     M15  ; 入料黏塵輪下降RY
      OUT     T21 D262  ; 入料黏塵輪下降T / 入料黏塵輪下降時間*10
1174  LDF     M16  ; 入料黏塵輪自動升降 RY
      OR      SM402  ; 初始脈波
      RST     M14  ; 入料黏塵輪上升RY
      RST     M15  ; 入料黏塵輪下降RY
1179  LD      X64  ; 出料網偏偵測(前)光電
      OUT     T46 K20  ; 出料網偏向前延遲
        [note] 
      AND     T46  ; 出料網偏向前延遲
      SET     M82  ; 出料網偏向前RY
      RST     M83  ; 出料網偏向後RY
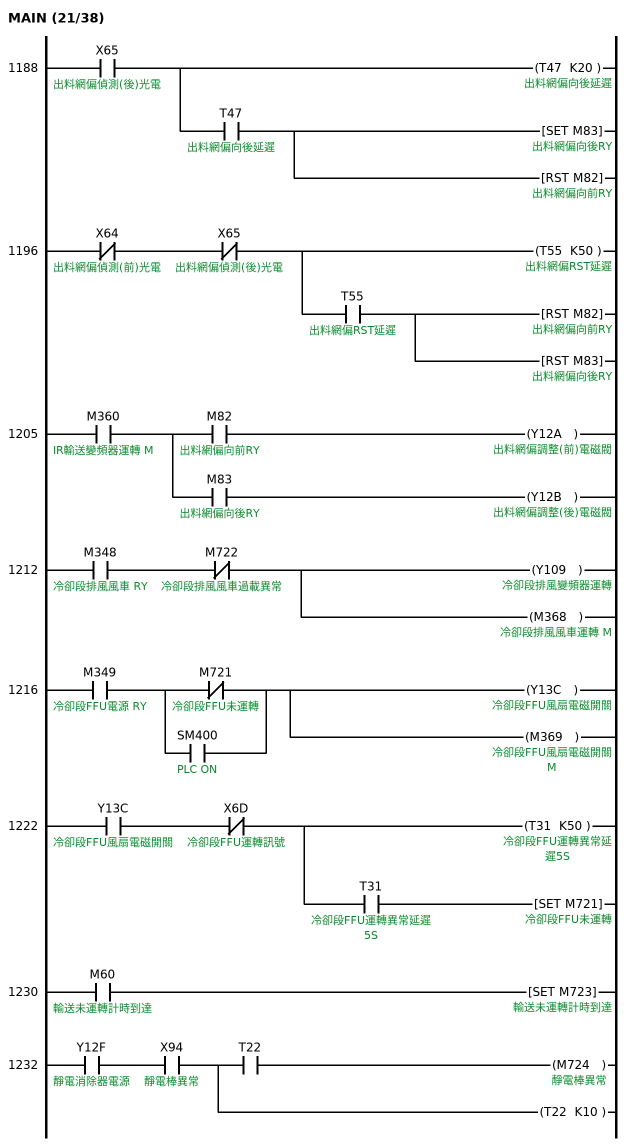
1188  LD      X65  ; 出料網偏偵測(後)光電
      OUT     T47 K20  ; 出料網偏向後延遲
      AND     T47  ; 出料網偏向後延遲
      SET     M83  ; 出料網偏向後RY
      RST     M82  ; 出料網偏向前RY
1196  LDI     X64  ; 出料網偏偵測(前)光電
      ANI     X65  ; 出料網偏偵測(後)光電
      OUT     T55 K50  ; 出料網偏RST延遲
      AND     T55  ; 出料網偏RST延遲
      RST     M82  ; 出料網偏向前RY
      RST     M83  ; 出料網偏向後RY
1205  LD      M360  ; IR輸送變頻器運轉 M
      MPS
      AND     M82  ; 出料網偏向前RY
      OUT     Y12A  ; 出料網偏調整(前)電磁閥
      MPP
      AND     M83  ; 出料網偏向後RY
      OUT     Y12B  ; 出料網偏調整(後)電磁閥
1212  LD      M348  ; 冷卻段排風風車 RY
      ANI     M722  ; 冷卻段排風風車過載異常
      OUT     Y109  ; 冷卻段排風變頻器運轉
      OUT     M368  ; 冷卻段排風風車運轉 M
1216  LD      M349  ; 冷卻段FFU電源 RY
      LDI     M721  ; 冷卻段FFU未運轉
      OR      SM400  ; PLC ON
      ANB
      OUT     Y13C  ; 冷卻段FFU風扇電磁開關
      OUT     M369  ; 冷卻段FFU風扇電磁開關 M
1222  LD      Y13C  ; 冷卻段FFU風扇電磁開關
      ANI     X6D  ; 冷卻段FFU運轉訊號
      OUT     T31 K50  ; 冷卻段FFU運轉異常延遲5S
      AND     T31  ; 冷卻段FFU運轉異常延遲5S
      SET     M721  ; 冷卻段FFU未運轉
1230  LD      M60  ; 輸送未運轉計時到達
      SET     M723  ; 輸送未運轉計時到達
1232  LD      Y12F  ; 靜電消除器電源
      AND     X94  ; 靜電棒異常
      MPS
      AND     T22
      OUT     M724  ; 靜電棒異常
      MPP
      OUT     T22 K10
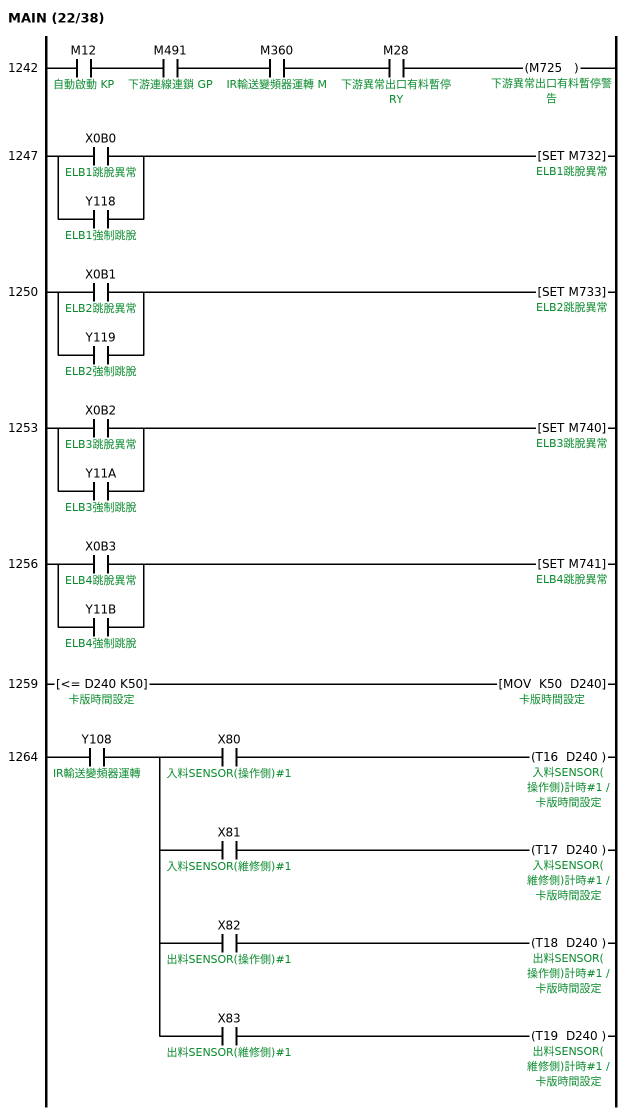
1242  LD      M12  ; 自動啟動 KP
      AND     M491  ; 下游連線連鎖 GP
      AND     M360  ; IR輸送變頻器運轉 M
      AND     M28  ; 下游異常出口有料暫停 RY
      OUT     M725  ; 下游異常出口有料暫停警告
1247  LD      X0B0  ; ELB1跳脫異常
      OR      Y118  ; ELB1強制跳脫
      SET     M732  ; ELB1跳脫異常
1250  LD      X0B1  ; ELB2跳脫異常
      OR      Y119  ; ELB2強制跳脫
      SET     M733  ; ELB2跳脫異常
1253  LD      X0B2  ; ELB3跳脫異常
      OR      Y11A  ; ELB3強制跳脫
      SET     M740  ; ELB3跳脫異常
1256  LD      X0B3  ; ELB4跳脫異常
      OR      Y11B  ; ELB4強制跳脫
      SET     M741  ; ELB4跳脫異常
1259  LD<=    D240 K50  ; 卡版時間設定
      MOV     K50 D240
1264  LD      Y108  ; IR輸送變頻器運轉
      MPS
      AND     X80  ; 入料SENSOR(操作側)#1
      OUT     T16 D240  ; 入料SENSOR(操作側)計時#1 / 卡版時間設定
      MRD
      AND     X81  ; 入料SENSOR(維修側)#1
      OUT     T17 D240  ; 入料SENSOR(維修側)計時#1 / 卡版時間設定
      MRD
      AND     X82  ; 出料SENSOR(操作側)#1
      OUT     T18 D240  ; 出料SENSOR(操作側)計時#1 / 卡版時間設定
      MPP
      AND     X83  ; 出料SENSOR(維修側)#1
      OUT     T19 D240  ; 出料SENSOR(維修側)計時#1 / 卡版時間設定
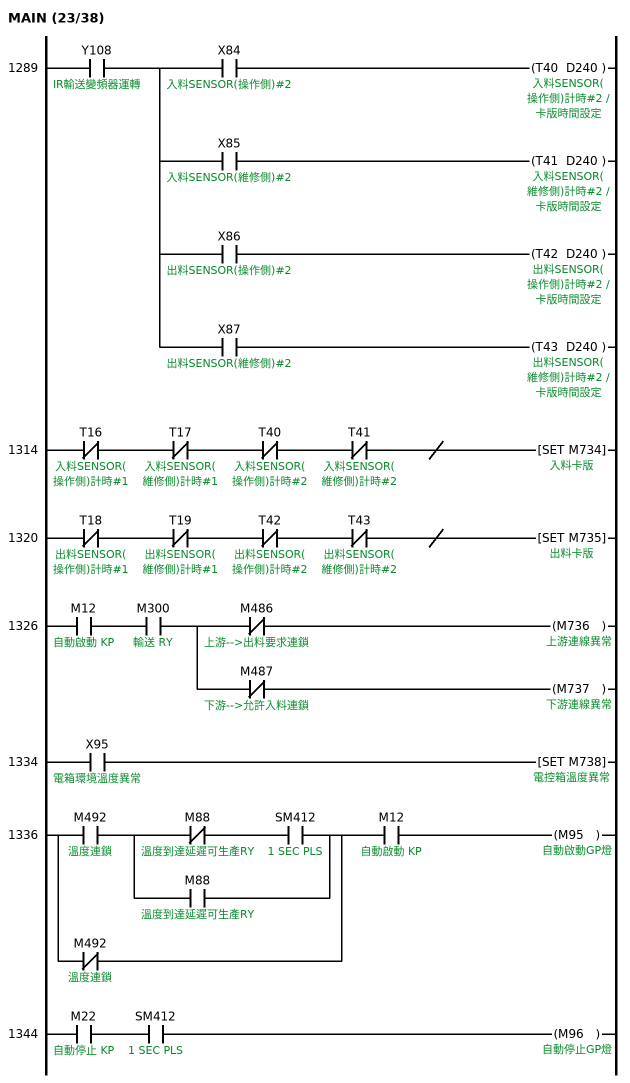
1289  LD      Y108  ; IR輸送變頻器運轉
      MPS
      AND     X84  ; 入料SENSOR(操作側)#2
      OUT     T40 D240  ; 入料SENSOR(操作側)計時#2 / 卡版時間設定
      MRD
      AND     X85  ; 入料SENSOR(維修側)#2
      OUT     T41 D240  ; 入料SENSOR(維修側)計時#2 / 卡版時間設定
      MRD
      AND     X86  ; 出料SENSOR(操作側)#2
      OUT     T42 D240  ; 出料SENSOR(操作側)計時#2 / 卡版時間設定
      MPP
      AND     X87  ; 出料SENSOR(維修側)#2
      OUT     T43 D240  ; 出料SENSOR(維修側)計時#2 / 卡版時間設定
1314  LDI     T16  ; 入料SENSOR(操作側)計時#1
      ANI     T17  ; 入料SENSOR(維修側)計時#1
      ANI     T40  ; 入料SENSOR(操作側)計時#2
      ANI     T41  ; 入料SENSOR(維修側)計時#2
      INV
      SET     M734  ; 入料卡版
1320  LDI     T18  ; 出料SENSOR(操作側)計時#1
      ANI     T19  ; 出料SENSOR(維修側)計時#1
      ANI     T42  ; 出料SENSOR(操作側)計時#2
      ANI     T43  ; 出料SENSOR(維修側)計時#2
      INV
      SET     M735  ; 出料卡版
1326  LD      M12  ; 自動啟動 KP
      AND     M300  ; 輸送 RY
      MPS
      ANI     M486  ; 上游-->出料要求連鎖
      OUT     M736  ; 上游連線異常
      MPP
      ANI     M487  ; 下游-->允許入料連鎖
      OUT     M737  ; 下游連線異常
1334  LD      X95  ; 電箱環境溫度異常
      SET     M738  ; 電控箱溫度異常
1336  LD      M492  ; 溫度連鎖
      LDI     M88  ; 溫度到達延遲可生產RY
      AND     SM412  ; 1 SEC PLS
      OR      M88  ; 溫度到達延遲可生產RY
      ANB
      ORI     M492  ; 溫度連鎖
      AND     M12  ; 自動啟動 KP
      OUT     M95  ; 自動啟動GP燈
1344  LD      M22  ; 自動停止 KP
      AND     SM412  ; 1 SEC PLS
      OUT     M96  ; 自動停止GP燈
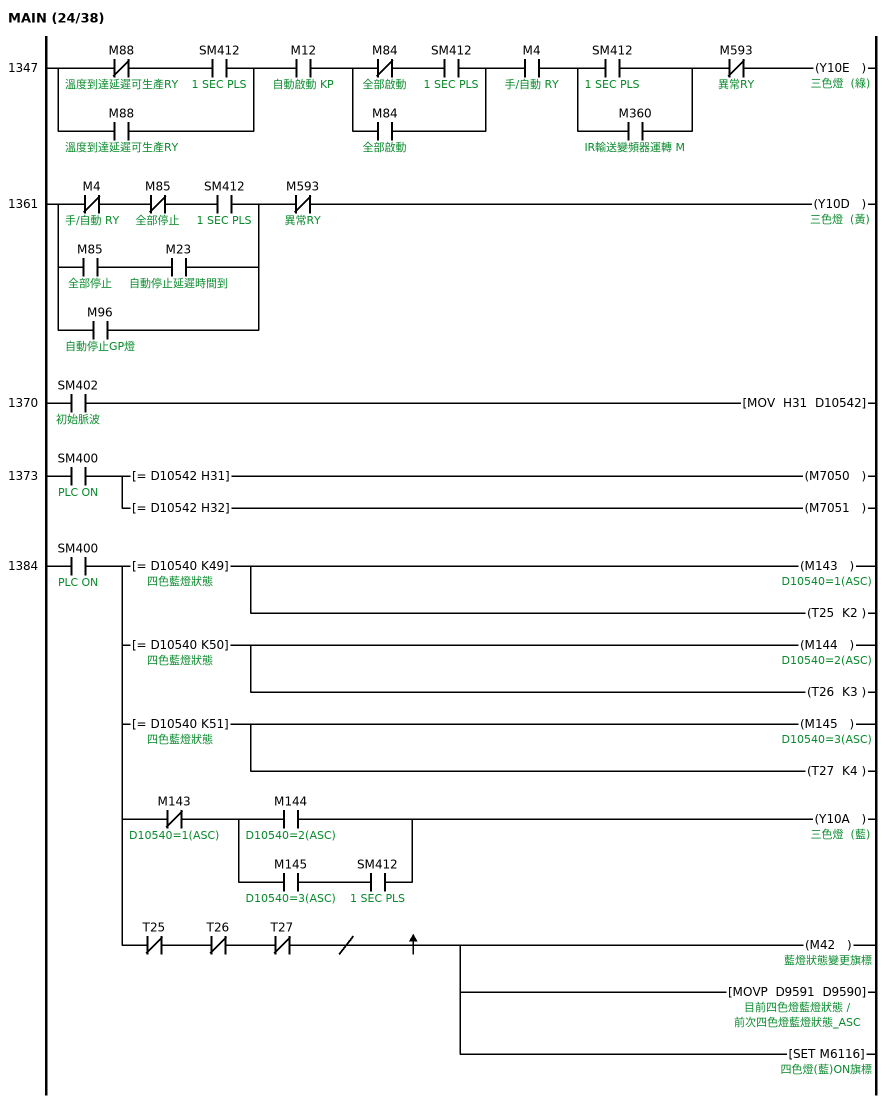
1347  LDI     M88  ; 溫度到達延遲可生產RY
      AND     SM412  ; 1 SEC PLS
      OR      M88  ; 溫度到達延遲可生產RY
      AND     M12  ; 自動啟動 KP
      LDI     M84  ; 全部啟動
      AND     SM412  ; 1 SEC PLS
      OR      M84  ; 全部啟動
      ANB
      AND     M4  ; 手/自動 RY
      LD      SM412  ; 1 SEC PLS
      OR      M360  ; IR輸送變頻器運轉 M
      ANB
      ANI     M593  ; 異常RY
      OUT     Y10E  ; 三色燈  (綠)
1361  LDI     M4  ; 手/自動 RY
      ANI     M85  ; 全部停止
      AND     SM412  ; 1 SEC PLS
      LD      M85  ; 全部停止
      AND     M23  ; 自動停止延遲時間到
      ORB
      OR      M96  ; 自動停止GP燈
      ANI     M593  ; 異常RY
      OUT     Y10D  ; 三色燈  (黃)
1370  LD      SM402  ; 初始脈波
      MOV     H31 D10542
1373  LD      SM400  ; PLC ON
      MPS
      AND=    D10542 H31
      OUT     M7050
      MPP
      AND=    D10542 H32
      OUT     M7051
1384  LD      SM400  ; PLC ON
      MPS
      AND=    D10540 K49  ; 四色藍燈狀態
      OUT     M143  ; D10540=1(ASC)
      OUT     T25 K2
      MRD
      AND=    D10540 K50  ; 四色藍燈狀態
      OUT     M144  ; D10540=2(ASC)
      OUT     T26 K3
      MRD
      AND=    D10540 K51  ; 四色藍燈狀態
      OUT     M145  ; D10540=3(ASC)
      OUT     T27 K4
      MRD
      ANI     M143  ; D10540=1(ASC)
      LD      M144  ; D10540=2(ASC)
      LD      M145  ; D10540=3(ASC)
      AND     SM412  ; 1 SEC PLS
      ORB
      ANB
      OUT     Y10A  ; 三色燈  (藍)
      MPP
      ANI     T25
      ANI     T26
      ANI     T27
      INV
      MEP
      OUT     M42  ; 藍燈狀態變更旗標
      MOVP    D9591 D9590  ; 目前四色燈藍燈狀態 / 前次四色燈藍燈狀態_ASC
      SET     M6116  ; 四色燈(藍)ON旗標
